Yaskawa INFORM job: ADD-TACK-BY-TEACH-IN.JBI

/JOB
//NAME ADD-TACK-BY-TEACH-IN
//POS
///NPOS 0,0,0,0,0,0
//INST
///DATE 2018/09/06 10:06
///ATTR SC,RW
///GROUP1 RB1,BS1
///GROUP2 ST1
NOP
END
